PROGRAM MAIN
VAR
	fbFixedPump1 : FB_FixedPump;
	fbAdjustPump2 : FB_AdjustablePump;
	
	fbController1 : FB_Controller(fbFixedPump1);
	fbController2 : FB_Controller(fbAdjustPump2);
	
	fNewRate : REAL := 40;
	
	bOn : BOOL;
	bOff : BOOL;
	
END_VAR

IF bOn THEN
	fbController1.bPumpOn := TRUE;
	fbController1.fNewRate := fNewRate;
	fbController2.bPumpOn := TRUE;
	fbController2.fNewRate := fNewRate;
END_IF
IF bOff THEN
	fbController1.bPumpOn := FALSE;
	fbController2.bPumpOn := FALSE;
	fbController1.bPumpOff := TRUE;
	fbController2.bPumpOff := TRUE;
	bOn := FALSE;
	bOff := FALSE;
END_IF


Act_CallingFB();

ACTION Act_CallingFB:
fbFixedPump1();
fbAdjustPump2();
fbController1();
fbController2();
END_ACTION

END_PROGRAM

(* stored: Version 1.1.0.1, ProductVersion 3.1.4024.16
   POU MAIN: Id {b539d5ca-b603-491f-8454-0265245e5a1d}, SpecialFunc None
   Action Act_CallingFB: Id {7a87845d-3944-465f-a122-b637fac10451} *)
